# EPICS substitutions: ipimbLib/Db/bldSettings.substitutions
file bldSettings.db
{
  pattern { "" }
  { "" }
}
